// TwinCAT 3 PLC project Development
// ProgramVersion: 3.1.4026.13
// CompilerDefines: release,VISU_USEPROPERTYINFO
// libraries:
//   Tc2_Drive, * (Beckhoff Automation GmbH)
//   Tc2_EtherCAT, * (Beckhoff Automation GmbH)
//   Tc2_MC2, * (Beckhoff Automation GmbH)
//   Tc2_MC2_Drive, * (Beckhoff Automation GmbH)
//   Tc2_Standard, * (Beckhoff Automation GmbH)
//   Tc2_System, * (Beckhoff Automation GmbH)
//   Tc2_Utilities, * (Beckhoff Automation GmbH)
//   Tc3_Element, * (Zerlauth)
//   Tc3_IPCDiag, * (Beckhoff Automation GmbH)
//   Tc3_Module, * (Beckhoff Automation GmbH)
// project tree:
//   GVLs/ IO.TcGVL (not stored)
//   InDevelopment/Axis/ FB_Axis.TcPOU, F_TcError.TcPOU (not stored), I_Axis.TcIO
//   InDevelopment/Contactor/ FB_Contactor.TcPOU
//   InDevelopment/Cylinder/ FB_Cylinder.TcPOU, ST_CylinderOptions.TcDUT (not stored)
//   InDevelopment/ FB_ComponentEX.TcPOU, FB_EthercatDiagnostic.TcPOU
//   InDevelopment/PnozMulti/ FB_PnozMulti.TcPOU
//   Modules/ FB_Module01.TcPOU, FB_Machine.TcPOU, FB_Module02.TcPOU
//   / PlcTask.TcTTO (not stored)
//   POUs/ FB_ComponentT.TcPOU, MAIN.TcPOU
// real-time tasks:
//   TASK PlcTask: cycle T#500ms, priority 21, ADS port 351
//   TASK UnitTestTask: cycle T#1ms, priority 1, ADS port 350
// motion (NC):
//   TASK NC-Task 1 SAF: cycle T#2ms, priority 4, ADS port 501
//   TASK NC-Task 1 SVB: cycle T#10ms, priority 8, ADS port 511
//   AXIS Achse 1 (id 1)
//     OtherSettings: AllowMotionCmdToSlave=true
//     encoder EncType=1
//     drive DrvType=5
//       Analog: TorqueSetpointScale=10, ScaleFactorActTorque=0.1
//       TimeComp: TaskDelayCycles=1
//     controller CtrType=1
//       CtrPara: PriorControlFactor=1
//         Observer: BandWidth=20
// I/O:
//   DEVICE Gerät 1 (EtherCAT) (disabled), AmsNetId 10.58.50.38.2.1
//     Klemme 1 (EK1100) [EK1100 EtherCAT-Koppler (2A E-Bus)]
//     Box 2 (EP1008-0001) [EP1008-0001 8 K. Dig. Eingang 24V, 3ms, M8]
// variable links:
//   Development/Development Instance <-> Device 1 (EtherCAT)
//     PlcTask Inputs/MAIN.fbMachine.fbEthercatDiagnostic.AmsNetID <-> InfoData/AmsNetId

// ---- InDevelopment/Axis/I_Axis.TcIO
INTERFACE I_Axis

METHOD PUBLIC M_Halt : BOOL
VAR_INPUT
END_VAR
END_METHOD

METHOD PUBLIC M_Home : BOOL
VAR_INPUT
	fPosition:					LREAL;
	eHomingMode:				MC_HomingMode;
	bClearPositionLag: 			BOOL;
END_VAR
END_METHOD

METHOD PUBLIC M_MoveAbsolute : BOOL
VAR_INPUT
	fPosition:				LREAL;
	fVelocity:				LREAL;
	fAcceleration:			LREAL:= 0.0;
	fDeceleration:			LREAL:= 0.0;
	fJerk:					LREAL:= 0.0;
END_VAR
END_METHOD

METHOD PUBLIC M_MoveRelative : BOOL
VAR_INPUT
	fDistance:				LREAL;
	fVelocity:				LREAL;
	fAcceleration:			LREAL:= 0.0;
	fDeceleration:			LREAL:= 0.0;
	fJerk:					LREAL:= 0.0;
END_VAR
END_METHOD

METHOD PUBLIC M_MoveVelocity : BOOL
VAR_INPUT
	fVelocity:				LREAL;
	fAcceleration:			LREAL:= 0.0;
	fDeceleration:			LREAL:= 0.0;
	fJerk:					LREAL:= 0.0;
END_VAR
END_METHOD

METHOD PUBLIC M_ReadBOOL : BOOL
VAR_INPUT
	 eParameterNumber:		MC_AxisParameter;		// MC_AxisParameter
	 bValue:				REFERENCE TO BOOL;
END_VAR
END_METHOD

METHOD PUBLIC M_ReadLREAL : BOOL
VAR_INPUT
	 eParameterNumber:		MC_AxisParameter;		// MC_AxisParameter
	 fValue:				REFERENCE TO LREAL;
END_VAR
END_METHOD

METHOD PUBLIC M_Reset : BOOL
VAR_INPUT
END_VAR
END_METHOD

METHOD PUBLIC M_SetPosition : BOOL
VAR_INPUT
	fPosition:					LREAL;
	bClearPositionLag: 			BOOL;
END_VAR
END_METHOD

METHOD PUBLIC M_WriteBOOL : BOOL
VAR_INPUT
	eParameterNumber:		MC_AxisParameter;		// MC_AxisParameter
	bPersistent:			BOOL;
	bValue:					BOOL;
END_VAR
END_METHOD

METHOD PUBLIC M_WriteLREAL : BOOL
VAR_INPUT
	eParameterNumber:		MC_AxisParameter;		// MC_AxisParameter
	bPersistent:			BOOL;
	fValue:					LREAL;
END_VAR
END_METHOD

END_INTERFACE

// ---- InDevelopment/Axis/FB_Axis.TcPOU
FUNCTION_BLOCK FB_Axis EXTENDS FB_Element IMPLEMENTS I_Axis
VAR_INPUT
END_VAR
VAR_OUTPUT
	stAxis:							AXIS_REF;
END_VAR
VAR
	stParameter:					ST_AxisParameterSet;
	stComponents:					ST_AxisComponents;
	
	// General
	fbPower: 						MC_Power;
	fbReset: 						MC_Reset;
	fbHome: 						MC_Home;

	// Motion function blocks
	fbJog:							MC_Jog;
	fbSetPosition: 					MC_SetPosition;
	fbMoveAbsolute: 				REFERENCE TO MC_MoveAbsolute := fbMoveAbsolute1;
	fbMoveAbsolute1: 				MC_MoveAbsolute;
	fbMoveAbsolute2: 				MC_MoveAbsolute;
	fbMoveVelocity: 				MC_MoveVelocity;
	fbMoveRelative: 				MC_MoveRelative;
	fbHalt: 						MC_Halt;
	fbStop: 						MC_Stop;
	
	// Read function blocks
	fbReadAxisComponents:			MC_ReadAxisComponents:= (Execute:= TRUE);	
	fbReadError: 					MC_ReadAxisError;
	fbReadParameterSet:				MC_ReadParameterSet:= (Execute:= TRUE);	
	fbReadBoolParameter:			MC_ReadBoolParameter;
	fbReadParameter: 				MC_ReadParameter;
	
	// Write function blocks                            		
	fbWriteBoolParameter: 			MC_WriteBoolParameter;
	fbWriteBoolParameterPersistent: MC_WriteBoolParameterPersistent;
	fbWriteParameter: 				MC_WriteParameter;
	fbWriteParameterPersistent: 	MC_WriteParameterPersistent;
END_VAR

// memcpy(adr(stAxis.NcToPlc.ErrorCode), adr(code), sizeof(stAxis.NcToPlc.ErrorCode));
SUPER^();

stAxis.ReadStatus();

fbPower(Axis:= stAxis);
	
fbReset(Axis:= stAxis);
fbReset.Execute:= FALSE;

fbJog(Axis:= stAxis);
IF NOT fbJog.Active THEN
	fbJog.Mode:= E_JogMode.MC_JOGMODE_STANDARD_SLOW;
END_IF
fbJog.JogForward:= FALSE;
fbJog.JogBackwards:= FALSE;

fbHome(Axis:= stAxis);
fbHome.Execute:= FALSE;
	
fbSetPosition(Axis:= stAxis);
fbSetPosition.Execute:= FALSE;

fbMoveAbsolute1(Axis:= stAxis);
fbMoveAbsolute1.Execute:= FALSE;
	
fbMoveAbsolute2(Axis:= stAxis);
fbMoveAbsolute2.Execute:= FALSE;
	
fbMoveRelative(Axis:= stAxis);
fbMoveRelative.Execute:= FALSE;
	
fbMoveVelocity(Axis:= stAxis);
fbMoveVelocity.Execute:= FALSE;

fbHalt(Axis:= stAxis);
fbHalt.Execute:= FALSE;
	
fbStop(Axis:= stAxis);
fbStop.Execute:= FALSE;
	
fbReadBoolParameter(Axis:= stAxis);
fbReadBoolParameter.Enable:= FALSE;

fbWriteBoolParameter(Axis:= stAxis);
fbWriteBoolParameter.Execute:= FALSE;

fbWriteBoolParameterPersistent(Axis:= stAxis);
fbWriteBoolParameterPersistent.Execute:= FALSE;

fbReadParameter(Axis:= stAxis);
fbReadParameter.Enable:= FALSE;
	
fbWriteParameter(Axis:= stAxis);
fbWriteParameter.Execute:= FALSE;

fbWriteParameterPersistent(Axis:= stAxis);
fbWriteParameterPersistent.Execute:= FALSE;
	
fbReadParameterSet(Parameter:=stParameter, Axis:= stAxis);
fbReadParameterSet.Execute:= FALSE;

fbReadAxisComponents(AxisComponents:= stComponents, Axis:= stAxis);
fbReadError(Axis:= stAxis, Enable:= TRUE);

METHOD PROTECTED M_Aborting : BOOL (* Return*)
M_Aborting:= TRUE;
END_METHOD

METHOD PROTECTED M_ErrorID
VAR_INPUT
	nErrorCode : UDINT;
END_VAR
IF nErrorCode >= 16#4000 AND nErrorCode <= 16#40FF THEN
		P_Event.M_AddSTRING(stParameter.sAxisName);
		P_Event.M_AddSTRING(F_TcError(nErrorCode));
		P_Event.M_Error('%s: General error (%s)',  1101);
	ELSIF nErrorCode >= 16#4100 AND nErrorCode <= 16#41FF THEN
		P_Event.M_AddSTRING(stParameter.sAxisName);
		P_Event.M_AddSTRING(F_TcError(nErrorCode));
		P_Event.M_Error('%s: Channel Errors (%s)',  1102);
	ELSIF nErrorCode >= 16#4200 AND nErrorCode <= 16#42FF THEN
		P_Event.M_AddSTRING(stParameter.sAxisName);
		P_Event.M_AddSTRING(F_TcError(nErrorCode));
		P_Event.M_Error('%s: Group error (%s)',  1103);
	ELSIF nErrorCode >= 16#4300 AND nErrorCode <= 16#43FF THEN
		P_Event.M_AddSTRING(stParameter.sAxisName);
		P_Event.M_AddSTRING(F_TcError(nErrorCode));
		P_Event.M_Error('%s: Axis error (%s)',  1104);
	ELSIF nErrorCode >= 16#4400 AND nErrorCode <= 16#44FF THEN
		P_Event.M_AddSTRING(stParameter.sAxisName);
		P_Event.M_AddSTRING(F_TcError(nErrorCode));
		P_Event.M_Error('%s: Encoder error (%s)',  1105);	
	ELSIF nErrorCode >= 16#4500 AND nErrorCode <= 16#45FF THEN
		P_Event.M_AddSTRING(stParameter.sAxisName);
		P_Event.M_AddSTRING(F_TcError(nErrorCode));
		P_Event.M_Error('%s: Controller error (%s)',  1106);	
	ELSIF nErrorCode >= 16#4600 AND nErrorCode <= 16#46FF THEN
		P_Event.M_AddSTRING(stParameter.sAxisName);
		P_Event.M_Error('%s: Drive error (%s)',  1107);	
	ELSIF nErrorCode >= 16#4A00 AND nErrorCode <= 16#4AFF THEN
		P_Event.M_AddSTRING(stParameter.sAxisName);
		P_Event.M_AddSTRING(F_TcError(nErrorCode));
		P_Event.M_Error('%s: Table error (%s)',  1108);	
	ELSIF nErrorCode >= 16#4B00 AND nErrorCode <= 16#4BFF THEN
		P_Event.M_AddSTRING(stParameter.sAxisName);
		P_Event.M_AddSTRING(F_TcError(nErrorCode));
		P_Event.M_Error('%s: NC PLC error (%s)',  1109);	
	ELSIF nErrorCode >= 16#4C00 AND nErrorCode <= 16#4CFF THEN
		P_Event.M_AddSTRING(stParameter.sAxisName);
		P_Event.M_AddSTRING(F_TcError(nErrorCode));
		P_Event.M_Error('%s: Kinematic Transformation (%s)',  1110);	
	ELSIF nErrorCode >= 16#8000 AND nErrorCode <= 16#8FFF THEN
		P_Event.M_AddSTRING(stParameter.sAxisName);
		P_Event.M_AddSTRING(F_TcError(nErrorCode));
		P_Event.M_Error('%s: NC error code extended (%s)',  1111);	
	ELSIF nErrorCode >= 16#8100 AND nErrorCode <= 16#81FF THEN
		P_Event.M_AddSTRING(stParameter.sAxisName);
		P_Event.M_AddSTRING(F_TcError(nErrorCode));
		P_Event.M_Error('%s: Bode plot (%s)',  1112);
	ELSIF nErrorCode >= 16#8200 AND nErrorCode <= 16#82FF THEN
		P_Event.M_AddSTRING(stParameter.sAxisName);
		P_Event.M_AddSTRING(F_TcError(nErrorCode));
		P_Event.M_Error('%s: Further errors (%s)',  1113);
	END_IF
END_METHOD

METHOD PROTECTED M_Execute : BOOL (* Return*)

M_Execute:= stAxis.Status.NotMoving and stAxis.Status.InTargetPosition;
END_METHOD

METHOD PUBLIC M_Halt : BOOL
VAR_INPUT
END_VAR
fbHalt.Execute:= TRUE;
M_Halt:= stAxis.Status.NotMoving;
END_METHOD

METHOD PUBLIC M_Home : BOOL
VAR_INPUT
	fPosition:					LREAL;
	eHomingMode:				MC_HomingMode;
	bClearPositionLag: 			BOOL;
END_VAR
fbHome.Execute:= TRUE;
fbHome.Position:= fPosition;
fbHome.HomingMode:= eHomingMode;
fbHome.Options.ClearPositionLag:= bClearPositionLag;
IF fbHome.Done THEN
	fbReset.Execute:= TRUE;
	M_Home:= TRUE;
END_IF
END_METHOD

METHOD PUBLIC M_MoveAbsolute : BOOL
VAR_INPUT
	fPosition:				LREAL;
	fVelocity:				LREAL;
	fAcceleration:			LREAL:= 0.0;
	fDeceleration:			LREAL:= 0.0;
	fJerk:					LREAL:= 0.0;
END_VAR
// Axis redy?
IF stAxis.Status.ControlLoopClosed THEN
	// input changed?
	IF fPosition <> fbMoveAbsolute.Position OR_ELSE fVelocity <> fbMoveAbsolute.Velocity OR_ELSE fbMoveAbsolute.Acceleration <> fbMoveAbsolute.Acceleration OR_ELSE fDeceleration <> fbMoveAbsolute.Deceleration OR_ELSE fJerk <> fbMoveAbsolute.Jerk THEN
		IF NOT fbMoveAbsolute1.Busy THEN
			// select axis 1
			fbMoveAbsolute:= fbMoveAbsolute1;
		ELSIF NOT fbMoveAbsolute2.Busy THEN
			// select axis 2
			fbMoveAbsolute:= fbMoveAbsolute2;
		ELSE
			// command blocked
			M_MoveAbsolute:= FALSE;
			RETURN;
		END_IF
		// take values
		fbMoveAbsolute.Execute:= 		TRUE;
		fbMoveAbsolute.Position:= 		fPosition;
		fbMoveAbsolute.Velocity:= 		fVelocity;
		fbMoveAbsolute.Acceleration:= 	fAcceleration;
		fbMoveAbsolute.Deceleration:= 	fDeceleration;
		fbMoveAbsolute.Jerk:= 			fJerk;
		M_MoveAbsolute:= FALSE;
	ELSE
		// Done
		M_MoveAbsolute:=  NOT (fbMoveAbsolute1.Active OR  NOT fbMoveAbsolute2.Active);
	END_IF
ELSE
	P_Event.M_AddSTRING(stParameter.sAxisName);
	P_Event.M_AddREAL(fPosition, 3);
	P_Event.M_AddREAL(fVelocity, 3);
	P_Event.M_Info('%s: Not ready for .M_MoveAbsolute(%s, %s)',  1114);
	M_MoveAbsolute:= FALSE;
END_IF
END_METHOD

METHOD PUBLIC M_MoveRelative : BOOL
VAR_INPUT
	fDistance:				LREAL;
	fVelocity:				LREAL;
	fAcceleration:			LREAL:= 0.0;
	fDeceleration:			LREAL:= 0.0;
	fJerk:					LREAL:= 0.0;
END_VAR
IF fbPower.Status THEN
	fbMoveRelative.Execute:= 			TRUE;
	fbMoveRelative.Distance:= 			fDistance;
	fbMoveRelative.Velocity:= 			fVelocity;
	fbMoveRelative.Acceleration:= 		fAcceleration;
	fbMoveRelative.Deceleration:= 		fDeceleration;
	fbMoveRelative.Jerk:= 				fJerk;
	M_MoveRelative:= 					fbMoveRelative.Done;
END_IF
END_METHOD

METHOD PUBLIC M_MoveVelocity : BOOL
VAR_INPUT
	fVelocity:				LREAL;
	fAcceleration:			LREAL:= 0.0;
	fDeceleration:			LREAL:= 0.0;
	fJerk:					LREAL:= 0.0;
END_VAR
IF fbPower.Status THEN
	fbMoveVelocity.Execute:= 			TRUE;
	fbMoveVelocity.Velocity:= 			fVelocity;
	fbMoveVelocity.Acceleration:= 		fAcceleration;
	fbMoveVelocity.Deceleration:= 		fDeceleration;
	fbMoveVelocity.Jerk:= 				fJerk;
	IF fVelocity >= 0.0 THEN
		fbMoveVelocity.Direction:= 			MC_Direction.MC_Positive_Direction;
	ELSE
		fbMoveVelocity.Direction:= 			MC_Direction.MC_Negative_Direction;	
	END_IF
	
	M_MoveVelocity:= fbMoveVelocity.InVelocity;
END_IF
END_METHOD

METHOD PUBLIC M_ReadBOOL : BOOL
VAR_INPUT
	 eParameterNumber:		MC_AxisParameter;		// MC_AxisParameter
	 bValue:				REFERENCE TO BOOL;
END_VAR
fbReadBoolParameter.Enable:= TRUE;
fbReadBoolParameter.ParameterNumber:= eParameterNumber;
fbReadBoolParameter.ReadMode:= E_ReadMode.READMODE_ONCE;
IF fbReadBoolParameter.Valid THEN
	IF __ISVALIDREF(bValue) THEN
		bValue:= fbReadBoolParameter.Value;
		M_ReadBOOL:= TRUE;		
	END_IF
END_IF
END_METHOD

METHOD PUBLIC M_ReadComponents : BOOL
VAR_INPUT
END_VAR
fbReadAxisComponents.Execute:= TRUE;
M_ReadComponents:= fbReadAxisComponents.Done;
END_METHOD

METHOD PUBLIC M_ReadLREAL : BOOL
VAR_INPUT
	 eParameterNumber:		MC_AxisParameter;		// MC_AxisParameter
	 fValue:				REFERENCE TO LREAL;
END_VAR
fbReadParameter.Enable:= TRUE;
fbReadParameter.ParameterNumber:= eParameterNumber;
fbReadParameter.ReadMode:= E_ReadMode.READMODE_ONCE;
IF fbReadParameter.Valid THEN
	IF __ISVALIDREF(fValue) THEN
		fValue:= fbReadParameter.Value;
		M_ReadLREAL:= TRUE;	
	END_IF
END_IF
END_METHOD

METHOD PUBLIC M_ReadParameterSet : BOOL
VAR_INPUT
END_VAR
fbReadParameterSet.Execute:= TRUE;
M_ReadParameterSet:= fbReadParameterSet.Done;
END_METHOD

METHOD PUBLIC M_Reset : BOOL
VAR_INPUT
END_VAR
fbReset.Execute:= TRUE;		
M_Reset:= TRUE;
END_METHOD

METHOD PROTECTED M_Resetting : BOOL (* Return state complete*)
fbReset.Execute:= TRUE;
M_ReadParameterSet();
M_ReadComponents();
M_Resetting:= TRUE;
END_METHOD

METHOD PROTECTED M_Running
IF stAxis.NcToPlc.ErrorCode <> 0 THEN
	M_ErrorID(stAxis.NcToPlc.ErrorCode);
END_IF
END_METHOD

METHOD PUBLIC M_SetPosition : BOOL
VAR_INPUT
	fPosition:					LREAL;
	bClearPositionLag: 			BOOL;
END_VAR
fbSetPosition.Execute:= TRUE;
fbSetPosition.Position:= fPosition;
fbSetPosition.Options.ClearPositionLag:= bClearPositionLag;
M_SetPosition:= fbSetPosition.Done;
END_METHOD

METHOD PROTECTED M_Starting : BOOL (* Return state complete*)
fbPower.Enable:= TRUE;
fbPower.Enable_Negative:= TRUE;
fbPower.Enable_Positive:= TRUE;
fbPower.Override:= 100.0;
fbPower.BufferMode:= MC_BufferMode.MC_Aborting;
M_Starting:= TRUE;
END_METHOD

METHOD PROTECTED M_Stopping : BOOL (* Return state complete*)
M_Stopping:= M_Halt();
END_METHOD

METHOD PUBLIC M_WriteBOOL : BOOL
VAR_INPUT
	eParameterNumber:		MC_AxisParameter;		// MC_AxisParameter
	bPersistent:			BOOL;
	bValue:					BOOL;
END_VAR
IF bPersistent THEN
	fbWriteBoolParameterPersistent.Execute:= TRUE;
	fbWriteBoolParameterPersistent.ParameterNumber:= eParameterNumber;
	fbWriteBoolParameterPersistent.Value:= bValue;
	IF fbWriteBoolParameterPersistent.Done THEN
		M_WriteBOOL:= TRUE;
	END_IF
ELSE
	fbWriteBoolParameter.Execute:= TRUE;
	fbWriteBoolParameter.ParameterNumber:= eParameterNumber;
	fbWriteBoolParameter.Value:= bValue;
	IF fbWriteBoolParameter.Done THEN
		M_WriteBOOL:= TRUE;
	END_IF
END_IF
END_METHOD

METHOD PUBLIC M_WriteLREAL : BOOL
VAR_INPUT
	eParameterNumber:		MC_AxisParameter;		// MC_AxisParameter
	bPersistent:			BOOL;
	fValue:					LREAL;
END_VAR
IF bPersistent THEN
	fbWriteParameterPersistent.Execute:= TRUE;
	fbWriteParameterPersistent.ParameterNumber:= eParameterNumber;
	fbWriteParameterPersistent.Value:= fValue;
	IF fbWriteParameterPersistent.Done THEN
		M_WriteLREAL:= TRUE;
	END_IF
ELSE
	fbWriteParameter.Execute:= TRUE;
	fbWriteParameter.ParameterNumber:= eParameterNumber;
	fbWriteParameter.Value:= fValue;
	IF fbWriteparameter.Done THEN
		M_WriteLREAL:= TRUE;
	END_IF
END_IF
END_METHOD

END_FUNCTION_BLOCK

// ---- InDevelopment/Contactor/FB_Contactor.TcPOU
FUNCTION_BLOCK FB_Contactor EXTENDS FB_Element
VAR_INPUT
	bInput				AT%I*: BOOL;
END_VAR
VAR_OUTPUT
	bOutput				AT%I*: BOOL;
END_VAR
VAR
END_VAR

super^();

METHOD PROTECTED M_Running
IF bOutput THEN
	IF bInput  THEN
		;
	ELSE
		P_Event.M_Abort('Feedback wrong state %s', 0);		
	END_IF
END_IF
END_METHOD

METHOD PROTECTED M_Starting : BOOL (* Return state complete*)
IF bOutput THEN
	IF bInput THEN
		M_Starting:= TRUE;
	ELSE
		P_Event.M_Abort('Feedback wrong state %s', 0);
	END_IF
ELSE
	IF bInput THEN
		P_Event.M_Abort('Feedback wrong state %s', 0);
	ELSE
		bOutput:= TRUE;
	END_IF	
	
END_IF
END_METHOD

END_FUNCTION_BLOCK

// ---- InDevelopment/Cylinder/FB_Cylinder.TcPOU
FUNCTION_BLOCK FB_Cylinder EXTENDS FB_Element
VAR_INPUT
	eEventType:				E_EventType:= E_EventType.Stop;
	stOptions:				ST_CylinderOptions;
END_VAR
VAR_OUTPUT
END_VAR
VAR
	bInHomePosition			AT%I*:		BOOL;
	bInWorkPosition			AT%I*:		BOOL;
	bToHomePosition			AT%Q*:		BOOL;
	bToWorkPosition			AT%Q*:		BOOL;
	fbHomePositon:			FB_Debounce;
	fbWorkPositon:			FB_Debounce;
	fbStarup:				TON;
	fbTimeout:				TON;
END_VAR

SUPER^();

METHOD PROTECTED M_Aborting : BOOL (* Return*)
bToHomePosition:= FALSE;
bToWorkPosition:= FALSE;
M_Aborting:= TRUE;
END_METHOD

METHOD PROTECTED M_Execute : BOOL // Return state complete
VAR_INPUT
END_VAR
fbHomePositon(bInput:= bInHomePosition);
fbWorkPositon(bInput:= bInWorkPosition);
fbTimeout(PT:= stOptions.tTimeout);
END_METHOD

METHOD PROTECTED M_Starting : BOOL // Return state complete
VAR_INPUT
END_VAR
IF SUPER^.M_Starting() THEN
	fbHomePositon.tTime:= stOptions.tDebounce;
	fbWorkPositon.tTime:= stOptions.tDebounce;
	// Check positons
	IF bToHomePosition AND bToWorkPosition THEN
		IF stOptions.tStartup <> T#0S THEN
			fbStarup(In:= TRUE, PT:= stOptions.tStartup);
			IF fbStarup.Q THEN
				fbStarup(In:= FALSE);
				bToHomePosition:= FALSE;
				bToWorkPosition:= FALSE;
				M_Starting:= TRUE;		
			END_IF
		ELSE
			M_Starting:= TRUE;	
		END_IF
	ELSIF bToHomePosition THEN
		IF NOT bInHomePosition THEN
			P_Event.M_AddSTRING(fbReflection.P_ID);
			P_Event.M_AddSTRING(stOptions.sHomePosition);
			P_Event.M_Error('Cylinder not in Home Positon (%s-%s)', 0);
		ELSIF bInWorkPosition THEN
			P_Event.M_AddSTRING(fbReflection.P_ID);
			P_Event.M_AddSTRING(stOptions.sWorkPosition);
			P_Event.M_Error('Cylinder in Work Positon (%s-%s)', 0);
		ELSE
			M_Starting:= TRUE;	
		END_IF
	ELSIF bToWorkPosition THEN
		IF NOT bInWorkPosition THEN
			P_Event.M_AddSTRING(fbReflection.P_ID);
			P_Event.M_AddSTRING(stOptions.sWorkPosition);
			P_Event.M_Error('Cylinder not in Work Positon (%s-%s)', 0);				
		ELSIF bInHomePosition THEN
			P_Event.M_AddSTRING(fbReflection.P_ID);
			P_Event.M_AddSTRING(stOptions.sHomePosition);
			P_Event.M_Error('Cylinder not in Home Positon (%s-%s)', 0);
		ELSE
			M_Starting:= TRUE;	
		END_IF
	ELSE
		IF bInWorkPosition THEN
			bToWorkPosition:= TRUE;
			M_Starting:= TRUE;
		ELSIF bInHomePosition THEN
			bToHomePosition:= TRUE;
			M_Starting:= TRUE;
		ELSIF stOptions.tStartup <> T#0S THEN		
			bToHomePosition:= TRUE;
			bToWorkPosition:= TRUE;
		ELSE
			M_Starting:= TRUE;
		END_IF
	END_IF
END_IF
END_METHOD

METHOD PUBLIC M_ToHome : BOOL
VAR_INPUT
END_VAR
IF bToWorkPosition THEN
	fbTimeout(IN:= FALSE);
	bToHomePosition:= TRUE;
	bToWorkPosition:= FALSE;

ELSIF bToHomePosition  THEN
	IF NOT fbWorkPositon.P_Value AND fbHomePositon.P_Value THEN
		M_ToHome:= TRUE;
	ELSE
		fbTimeout.IN:= TRUE;
		IF fbTimeout.Q THEN
			IF fbWorkPositon.P_Value THEN
				CASE eEventType OF
					E_EventType.Information:
						P_Event.M_AddSTRING(fbReflection.P_ID);
						P_Event.M_AddSTRING(stOptions.sWorkPosition);
						P_Event.M_Info('Cylinder Work Positon not left (%s%s)', 1120);	
					E_EventType.Warning:
						P_Event.M_AddSTRING(fbReflection.P_ID);
						P_Event.M_AddSTRING(stOptions.sWorkPosition);
						P_Event.M_Warning('Cylinder Work Positon not left (%s%s)', 1120);						
					E_EventType.Stop:
						P_Event.M_AddSTRING(fbReflection.P_ID);
						P_Event.M_AddSTRING(stOptions.sWorkPosition);
						P_Event.M_Error('Cylinder Work Positon not left (%s%s)', 1120);				
					E_EventType.Abort:				
						P_Event.M_AddSTRING(fbReflection.P_ID);
						P_Event.M_AddSTRING(stOptions.sWorkPosition);
						P_Event.M_Abort('Cylinder Work Positon not left (%s%s)', 1120);							
				END_CASE

			ELSIF NOT fbHomePositon.P_Value THEN
				CASE eEventType OF
					E_EventType.Information:
						P_Event.M_AddSTRING(fbReflection.P_ID);
						P_Event.M_AddSTRING(stOptions.sHomePosition);
						P_Event.M_Info('Cylinder Home Positon not reached (%s%s)', 1121);
					E_EventType.Warning:
						P_Event.M_AddSTRING(fbReflection.P_ID);
						P_Event.M_AddSTRING(stOptions.sHomePosition);
						P_Event.M_Warning('Cylinder Home Positon not reached (%s%s)', 1121);				
					E_EventType.Stop:
						P_Event.M_AddSTRING(fbReflection.P_ID);
						P_Event.M_AddSTRING(stOptions.sWorkPosition);
						P_Event.M_Error('Cylinder Home Positon not reached (%s%s)', 1121);		
					E_EventType.Abort:				
						P_Event.M_AddSTRING(fbReflection.P_ID);
						P_Event.M_AddSTRING(stOptions.sHomePosition);
						P_Event.M_Abort('Cylinder Home Positon not reached (%s%s)', 1121);
				END_CASE
				
			END_IF
		END_IF
	END_IF
END_IF
END_METHOD

METHOD PUBLIC M_ToWork : BOOL
VAR_INPUT
END_VAR
IF bToHomePosition THEN
	fbTimeout(IN:= FALSE);
	bToHomePosition:= FALSE;
	bToWorkPosition:= TRUE;	

ELSIF bToWorkPosition  THEN
	IF fbWorkPositon.P_Value AND NOT fbHomePositon.P_Value THEN
		M_ToWork:= TRUE;
	ELSE
		fbTimeout.IN:= TRUE;
		IF fbTimeout.Q THEN
			IF NOT fbWorkPositon.P_Value THEN
				CASE eEventType OF
					E_EventType.Information:
						P_Event.M_AddSTRING(fbReflection.P_ID);
						P_Event.M_AddSTRING(stOptions.sWorkPosition);
						P_Event.M_Info('Cylinder Work Positon not reached (%s%s)', 1122);	
					E_EventType.Warning:
						P_Event.M_AddSTRING(fbReflection.P_ID);
						P_Event.M_AddSTRING(stOptions.sWorkPosition);
						P_Event.M_Warning('Cylinder Work Positon not reached (%s%s)', 1122);						
					E_EventType.Stop:
						P_Event.M_AddSTRING(fbReflection.P_ID);
						P_Event.M_AddSTRING(stOptions.sWorkPosition);
						P_Event.M_Error('Cylinder Work Positon not reached (%s%s)', 1122);				
					E_EventType.Abort:				
						P_Event.M_AddSTRING(fbReflection.P_ID);
						P_Event.M_AddSTRING(stOptions.sWorkPosition);
						P_Event.M_Abort('Cylinder Work Positon not reached (%s%s)', 1122);							
				END_CASE

			ELSIF fbHomePositon.P_Value THEN
				CASE eEventType OF
					E_EventType.Information:
						P_Event.M_AddSTRING(fbReflection.P_ID);
						P_Event.M_AddSTRING(stOptions.sHomePosition);
						P_Event.M_Info('Cylinder Home Positon not left (%s%s)', 1122);
					E_EventType.Warning:
						P_Event.M_AddSTRING(fbReflection.P_ID);
						P_Event.M_AddSTRING(stOptions.sHomePosition);
						P_Event.M_Warning('Cylinder Home Positon not left (%s%s)', 1122);				
					E_EventType.Stop:
						P_Event.M_AddSTRING(fbReflection.P_ID);
						P_Event.M_AddSTRING(stOptions.sWorkPosition);
						P_Event.M_Error('Cylinder Home Positon not left (%s%s)', 1122);		
					E_EventType.Abort:				
						P_Event.M_AddSTRING(fbReflection.P_ID);
						P_Event.M_AddSTRING(stOptions.sHomePosition);
						P_Event.M_Abort('Cylinder Home Positon not left (%s%s)', 1122);
				END_CASE
				
			END_IF
		END_IF
	END_IF
END_IF
END_METHOD

{attribute 'suppress_wrn_C0410'}
PROPERTY PUBLIC P_Options : REFERENCE TO ST_CylinderOptions
GET
P_Options ref= stOptions;
END_GET
END_PROPERTY

END_FUNCTION_BLOCK

// ---- InDevelopment/FB_ComponentEX.TcPOU
FUNCTION_BLOCK FB_ComponentEX EXTENDS FB_Element
VAR_INPUT
END_VAR
VAR_OUTPUT
END_VAR
VAR
	bError:			BOOL;
	bAbort:			BOOL;
	bStop:			BOOL;
	bInformation:	BOOL;
	bWarning:		BOOL;
END_VAR

SUPER^();

METHOD PROTECTED M_Execute : BOOL
VAR_INPUT
END_VAR
CASE fbSequence.P_Number OF
	E_Sequence.Start:
		fbSequence.M_Await('Start', 0, T#0S, T#0S, TRUE, TRUE, 10);
	
	10:
		fbSequence.M_Await('Step 10',0,  T#0S, T#0S, TRUE, TRUE, 20);
		
	20:
		fbSequence.M_Await('Step 20',0,  T#0S, T#0S, FALSE, TRUE, E_Sequence.Done);	
		
	E_Sequence.Done:
		fbSequence.M_Reset();
		
END_CASE

IF bAbort THEN
	bAbort:= FALSE;
	fbEvent.M_AddSTRING('1');
	fbEvent.M_AddSTRING('2');
	fbEvent.M_AddSTRING('3');
	fbEvent.M_Abort('First Error Abort %s %s %s', 6);
END_IF

IF bStop THEN
	bStop:= FALSE;
	fbEvent.M_AddSTRING('a');
	fbEvent.M_AddSTRING('b');
	fbEvent.M_AddSTRING('c');
	fbEvent.M_Error('First Error Stop', 7);
END_IF

IF bInformation THEN
	fbEvent.M_Info('Info', 12);	
END_IF

IF bWarning THEN
	fbEvent.M_Warning('Warning', 13);	
END_IF
END_METHOD

END_FUNCTION_BLOCK

// ---- InDevelopment/FB_EthercatDiagnostic.TcPOU
FUNCTION_BLOCK FB_EthercatDiagnostic
VAR_GENERIC CONSTANT
    nLength				AT%I*:	UINT:= 100;
END_VAR
VAR_INPUT
	AmsNetID					AT%I*: AmsNetID;
END_VAR
VAR_OUTPUT
END_VAR
VAR_IN_OUT
END_VAR
VAR
	sNetId:						T_AmsNetId;					// Internal netid as string
	fbGetMasterState:			FB_EcGetMasterState;		// Get Master State
	fbGetMasterFrameStatistic:	FB_EcMasterFrameStatistic; 
	fbGetSlaveAddresses: 		FB_EcGetAllSlaveAddr;		// Get Slave Addresses
	fbGetAllSlaveStates:		FB_EcGetAllSlaveStates;		// Get Slave States
	fbGetSlaveCount:			FB_EcGetSlaveCount;
	fbGetScannedSlaves:			FB_EcGetScannedSlaves;		// Scan Slaves
	fbGetSlaveIdentity:			FB_EcGetSlaveIdentity;		// Get Slave Identities
	nState:						INT;
	aSlaveAdress:				ARRAY[0..nLength-1] OF UINT;
	aSlaveState:				ARRAY[0..nLength-1] OF ST_EcSlaveState;
	aSlaveScanned:				ARRAY[0..nLength-1] OF ST_EcSlaveScannedData;
END_VAR



CASE nState OF
	0: 
		sNetId:= F_CreateAmsNetId(AmsNetID);
		IF sNetId <> '0.0.0.0.0.0' THEN
			nState:= 10;
		END_IF
		
	10:
		IF M_GetMasterState() THEN
			nState:= 20;
		END_IF
		
	20:
		IF M_GetSlaveAdresses() THEN
			nState:= 30;
		END_IF
		
	30:
		IF M_GetScannedSlaves() THEN
			nState:= 40;
		END_IF
		
	40:
	
END_CASE

fbGetMasterState(sNetId:= sNetId);
fbGetMasterState.bExecute:= FALSE;

fbGetMasterFrameStatistic(sNetId:= sNetId);
fbGetMasterFrameStatistic.bExecute:= FALSE;

fbGetSlaveAddresses(sNetId:= sNetId);
fbGetSlaveAddresses.bExecute:= FALSE;

fbGetAllSlaveStates(sNetId:= sNetId);
fbGetAllSlaveStates.bExecute:= FALSE;

fbGetSlaveCount(sNetId:= sNetId);
fbGetSlaveCount.bExecute:= FALSE;

fbGetScannedSlaves(sNetId:= sNetId);
fbGetScannedSlaves.bExecute:= FALSE;

fbGetSlaveIdentity(sNetId:= sNetId);
fbGetSlaveIdentity.bExecute:= FALSE;

METHOD M_GetMasterFrameStatistic : BOOL
VAR_INPUT
END_VAR
IF fbGetMasterFrameStatistic.bExecute THEN
	IF fbGetMasterFrameStatistic.bBusy THEN
		;
	ELSIF fbGetMasterFrameStatistic.bError THEN
		;
	ELSE
		fbGetMasterFrameStatistic.bExecute:= FALSE;
		M_GetMasterFrameStatistic:= TRUE;
	END_IF

ELSE
	fbGetMasterFrameStatistic.bExecute:= TRUE;
END_IF
END_METHOD

METHOD PROTECTED M_GetMasterState : BOOL
VAR_INPUT
END_VAR
IF fbGetMasterState.bExecute THEN
	IF fbGetMasterState.bBusy THEN
		;
	ELSIF fbGetMasterState.bError THEN
		;
	ELSE
		fbGetMasterState.bExecute:= FALSE;
		M_GetMasterState:= TRUE;
	END_IF

ELSE
	fbGetMasterState.bExecute:= TRUE;
END_IF
END_METHOD

METHOD PROTECTED M_GetScannedSlaves : BOOL
VAR_INPUT
END_VAR
IF fbGetScannedSlaves.bExecute THEN
	IF fbGetScannedSlaves.bBusy THEN
		;
	ELSIF fbGetScannedSlaves.bError THEN
		;
	ELSE
		fbGetScannedSlaves.bExecute:= FALSE;
		M_GetScannedSlaves:= TRUE;
	END_IF
ELSE
	fbGetScannedSlaves.bExecute:= TRUE;
	fbGetScannedSlaves.pArrEcScannedSlaveInfo:= ADR(aSlaveScanned);
	fbGetScannedSlaves.cbBufLen:= SIZEOF(aSlaveScanned);
END_IF
END_METHOD

METHOD PROTECTED M_GetSlaveAdresses : BOOL
VAR_INPUT
END_VAR
IF fbGetSlaveAddresses.bExecute THEN
	IF fbGetSlaveAddresses.bBusy THEN
		;
	ELSIF fbGetSlaveAddresses.bError THEN
		;
	ELSE
		fbGetSlaveAddresses.bExecute:= FALSE;
		M_GetSlaveAdresses:= TRUE;
	END_IF

ELSE
	fbGetSlaveAddresses.bExecute:= TRUE;
	fbGetSlaveAddresses.pAddrBuf:= ADR(aSlaveAdress);
	fbGetSlaveAddresses.cbBufLen:= SIZEOF(aSlaveAdress);
END_IF
END_METHOD

METHOD PROTECTED M_GetSlaveCount : BOOL
VAR_INPUT
END_VAR
IF fbGetSlaveCount.bExecute THEN
	IF fbGetSlaveCount.bBusy THEN
		;
	ELSIF fbGetSlaveCount.bError THEN
		;
	ELSE
		fbGetSlaveCount.bExecute:= FALSE;
		M_GetSlaveCount:= TRUE;
	END_IF

ELSE
	fbGetSlaveCount.bExecute:= TRUE;
END_IF
END_METHOD

METHOD PROTECTED M_GetSlaveIdentity : BOOL
VAR_INPUT
	nSlaveAddress:			UINT;		
END_VAR
IF fbGetSlaveIdentity.bExecute THEN
	IF fbGetSlaveIdentity.bBusy AND NOT fbGetSlaveIdentity.bError THEN
		;
	ELSE
		fbGetSlaveIdentity.bExecute:= FALSE;
		M_GetSlaveIdentity:= TRUE;
	END_IF

ELSE
	fbGetSlaveIdentity.bExecute:= TRUE;
	fbGetSlaveIdentity.nSlaveAddr:= nSlaveAddress;
END_IF
END_METHOD

METHOD PROTECTED M_GetSlaveStates : BOOL
VAR_INPUT
END_VAR
IF fbGetAllSlaveStates.bExecute THEN
	IF fbGetAllSlaveStates.bBusy THEN
		;
	ELSIF fbGetAllSlaveStates.bError THEN
		;
	ELSE
		fbGetAllSlaveStates.bExecute:= FALSE;
		M_GetSlaveStates:= TRUE;
	END_IF

ELSE
	fbGetAllSlaveStates.bExecute:= TRUE;
	fbGetAllSlaveStates.pStateBuf:= ADR(aSlaveState);
	fbGetAllSlaveStates.cbBufLen:= SIZEOF(aSlaveState);
END_IF
END_METHOD

END_FUNCTION_BLOCK

// ---- InDevelopment/PnozMulti/FB_PnozMulti.TcPOU
FUNCTION_BLOCK FB_PnozMulti EXTENDS FB_Element
VAR_INPUT
END_VAR
VAR_OUTPUT
END_VAR
VAR
	bOK:					BOOL:= TRUE;
	bReset:					BOOL;
	fbReset:				TON:= (PT:= T#1S);
END_VAR

SUPER^();

METHOD PROTECTED M_Resetting : BOOL // Return state complete
VAR_INPUT
END_VAR
SUPER^.M_Resetting();
bReset:= TRUE;
fbReset(IN:= TRUE, PT:= T#1S);
IF fbReset.Q THEN
	bReset:= FALSE;
	M_Resetting:= TRUE;
END_IF
END_METHOD

METHOD PROTECTED M_Running
IF NOT bOK THEN
	P_Event.M_AddSTRING(fbReflection.P_ID);
	P_Event.M_Abort('PnozMulti no ok Signal (%s)', 0);
END_IF
END_METHOD

END_FUNCTION_BLOCK

// ---- Modules/FB_Module01.TcPOU
FUNCTION_BLOCK FB_Module01 EXTENDS FB_Module
VAR_INPUT
END_VAR
VAR_OUTPUT
END_VAR
VAR
END_VAR

// https://peterzerlauth.com/
SUPER^();

METHOD PROTECTED M_Execute : BOOL
VAR_INPUT
END_VAR
VAR
	bReturn:					BOOL:= TRUE;
END_VAR
M_Execute:= TRUE;
END_METHOD

METHOD PROTECTED M_Running
VAR_INPUT
END_VAR
END_METHOD

METHOD PROTECTED M_Starting : BOOL
VAR_INPUT
END_VAR
M_Starting:= SUPER^.M_Starting();
END_METHOD

METHOD PROTECTED M_Stopping : BOOL // Return state complete
VAR_INPUT
END_VAR
// State Stopping
M_Stopping:= SUPER^.M_Stopping();
END_METHOD

END_FUNCTION_BLOCK

// ---- Modules/FB_Machine.TcPOU
FUNCTION_BLOCK FB_Machine EXTENDS FB_Module
VAR_INPUT
END_VAR
VAR_OUTPUT
END_VAR
VAR
	fbEthercatDiagnostic:	FB_EthercatDiagnostic<10>;
END_VAR

// https://peterzerlauth.com/

fbEthercatDiagnostic();

SUPER^();

METHOD PROTECTED M_Execute : BOOL
VAR_INPUT
END_VAR
VAR
	bReturn:					BOOL:= TRUE;
END_VAR
M_Execute:= TRUE;
END_METHOD

METHOD PROTECTED M_Starting : BOOL
VAR_INPUT
END_VAR
M_Starting:= SUPER^.M_Starting();
END_METHOD

METHOD PROTECTED M_Stopping : BOOL // Return state complete
VAR_INPUT
END_VAR
// State Stopping
M_Stopping:= SUPER^.M_Stopping();
END_METHOD

END_FUNCTION_BLOCK

// ---- Modules/FB_Module02.TcPOU
FUNCTION_BLOCK FB_Module02 EXTENDS FB_Module
VAR_INPUT
END_VAR
VAR_OUTPUT
END_VAR
VAR
	fbPnozMulti:				FB_PnozMulti;
	fbComponent0:				FB_ComponentEx;
	fbComponent1:				FB_ComponentEx;
	fbContactor:				FB_Contactor;
	fbCylinder:					FB_Cylinder;
END_VAR

// https://peterzerlauth.com/
SUPER^();

fbComponent0();
fbComponent1();
fbContactor();
fbCylinder();
fbPnozMulti();

fbContactor.bInput:= fbContactor.bOutput;

METHOD PROTECTED M_Execute : BOOL
VAR_INPUT
END_VAR
VAR
	bReturn:					BOOL:= TRUE;
END_VAR
CASE fbSequence.P_Number OF
	E_Sequence.Start:
		bReturn:= TRUE;
		fbSequence.M_Await('Start 0', 0,  T#0S , T#1S, TRUE, bReturn, 10);
	
	10:
		bReturn:= TRUE;
		fbSequence.M_Await('Step 10', 0,  T#0S, T#0S, TRUE, bReturn, 20);
		
	20:
		bReturn:= TRUE;
		fbSequence.M_Await('Step 20', 0,  T#1S, T#0S, FALSE, bReturn, E_Sequence.Done);
		IF fbSequence.P_Timeout THEN
			fbEvent.M_Error('Overrride timeout error', 0);
		END_IF
		
	E_Sequence.Done:
		fbSequence.M_Reset();

END_CASE
END_METHOD

METHOD PROTECTED M_Idle : BOOL (* Return*)
SUPER^.M_Idle();

fbLevel4.M_Attach(fbPnozMulti);

fbLevel3.M_Attach(fbComponent0);
fbLevel3.M_Attach(fbComponent1);

fbLevel2.M_Attach(fbPnozMulti);
fbLevel2.M_Attach(fbContactor);

fbLevel1.M_Attach(fbCylinder);
END_METHOD

END_FUNCTION_BLOCK

// ---- POUs/FB_ComponentT.TcPOU
FUNCTION_BLOCK FB_ComponentT EXTENDS FB_Element
VAR_INPUT
END_VAR
VAR_OUTPUT
END_VAR
VAR
	bAbort: BOOL;
END_VAR

super^();

METHOD PROTECTED M_Execute : BOOL (* Return*)

IF bAbort THEN
	P_Event.M_Abort('msg', 0);
END_IF
END_METHOD

END_FUNCTION_BLOCK

// ---- POUs/MAIN.TcPOU
PROGRAM MAIN
VAR
	bTest:				BOOL;
	fbMachine:			FB_Machine;
	fbModule1:			FB_Module01;
	fbModule2:			FB_Module02;
	
	fbComponent1:		FB_ComponentT;
	fbComponent2:		FB_ComponentT;	
	bInit: 				BOOL:= TRUE;
	exceptionCode: 		__SYSTEM.ExceptionCode;
	exception: 			__SYSTEM.ExceptionCode;
	fbFileLogger:		FB_FileLogger<10>:= (sPathName:= 'C:\temp\log.txt');
END_VAR

bTest:= NOT bTest;

__TRY
	fbMachine();
	fbModule1();
	fbModule2();


	fbComponent1();
	fbComponent2();
__CATCH(exceptionCode)
 exception:= exceptionCode;
__ENDTRY




IF bInit THEN
	bInit:= False;
	fbComponent1.P_Event.P_Observer.M_Attach(fbComponent2);
	fbComponent2.P_Event.P_Observer.M_Attach(fbComponent1);
END_IF


fbFileLogger();

END_PROGRAM
